FUNCTION_BLOCK Test_TStringSplitter_ReturnsRemainder EXTENDS T_UnitTestBase
VAR
    StringSplitter : T_StringSplitter;
END_VAR

{attribute 'analysis' := '-33'} // inhibit unused variable warning
METHOD RunTest
IF Retest THEN
	SUPER^.Init();
END_IF

IF TestCompleted THEN
	RETURN;
END_IF


StringSplitter.Init(Str    := 'Bob$TCharles$TDavid',
                    Delim1 := '$T',
                    Delim2 := '');

AssertEquals_BOOL(Expected := TRUE,
                  Actual   := StringSplitter.HasMore(),
                  Message  := 'StringSplitter.HasMore()');

AssertEquals_STRING(Expected := 'Bob',
                    Actual   := StringSplitter.GetNext(),
                    Message  := 'StringSplitter.GetNext()');

AssertEquals_STRING(Expected := 'Charles$TDavid',
                    Actual   := StringSplitter.GetRemainder(),
                    Message  := 'StringSplitter.GetRemainder()');

AssertEquals_STRING(Expected := '',
                    Actual   := StringSplitter.GetRemainder(),
                    Message  := 'StringSplitter.GetRemainder()');

AssertEquals_BOOL(Expected := FALSE,
                  Actual   := StringSplitter.HasMore(),
                  Message  := 'StringSplitter.HasMore()');

TestCompleted := TRUE;
END_METHOD

END_FUNCTION_BLOCK

(* stored: Version 1.1.0.1, ProductVersion 3.1.4024.12
   POU Test_TStringSplitter_ReturnsRemainder: Id {8f4fe42a-2bd0-0874-1c8d-73d72a974ba0}, SpecialFunc None
   Method RunTest: Id {d7cd6f02-0e90-0914-1849-dc83b7fa3ea2} *)
